FUNCTION_BLOCK T_AdsReadWrite
VAR_INPUT
END_VAR
VAR_OUTPUT
END_VAR
VAR
    AdsReadWrite : ADSRDWRT;
    _Execution   : T_Execution;
END_VAR

IF _Execution.Aborting THEN
    _Execution.SetAborted();
END_IF

AdsReadWrite(NETID    :=,
             PORT     :=,
             IDXGRP   :=,
             IDXOFFS  :=,
             WRITELEN :=,
             READLEN  :=,
             SRCADDR  :=,
             DESTADDR :=,
             WRTRD    := _Execution.Starting,
             TMOUT    :=,
             BUSY     =>,
             ERR      =>,
             ERRID    =>);

IF _Execution.Starting THEN
    _Execution.SetBusy();
END_IF
IF _Execution.Busy AND NOT AdsReadWrite.BUSY THEN
    IF AdsReadWrite.ERR THEN
        _Execution.SetError(F_ErrorIdToString(AdsReadWrite.ERRID));
    ELSE
        _Execution.SetDone();
    END_IF
END_IF

METHOD Execute : BOOL
VAR_INPUT
    AmsNetId           : T_AmsNetID;
    Port               : T_AmsPort;
    IndexGroup         : UDINT;
    IndexOffset        : UDINT;
    ArgsAddress        : PVOID;
    ArgsLength         : UDINT;
    ReturnValueAddress : PVOID;
    ReturnValueLength  : UDINT;
END_VAR
IF _Execution.Start() THEN
    AdsReadWrite.NETID   := AmsNetId;
    AdsReadWrite.PORT    := Port;
    AdsReadWrite.IDXGRP  := IndexGroup;
    AdsReadWrite.IDXOFFS := IndexOffset;
    // Data to be written...
    AdsReadWrite.SRCADDR  := ArgsAddress;
    AdsReadWrite.WRITELEN := ArgsLength;
    // Data returned...
    AdsReadWrite.DESTADDR := ReturnValueAddress;
    AdsReadWrite.READLEN  := ReturnValueLength;
END_IF
END_METHOD

PROPERTY Execution : I_Execution
GET
Execution := _Execution;
END_GET
END_PROPERTY

END_FUNCTION_BLOCK

(* stored: Version 1.1.0.1, ProductVersion 3.1.4024.12
   POU T_AdsReadWrite: Id {5aec252a-cd25-0680-3f48-2fefdad531b3}, SpecialFunc None
   Method Execute: Id {3b6f6d27-4076-0e86-0c12-92bfcd385060}
   Property Execution: Id {c61d60c8-81bd-0935-03bc-90d31f301497}
   Get Get: Id {e1cd9cd8-1459-05e8-1090-07b0ed11fde2} *)
